PROGRAM Control_FBD
VAR

	timeStop: BOOL;
END_VAR

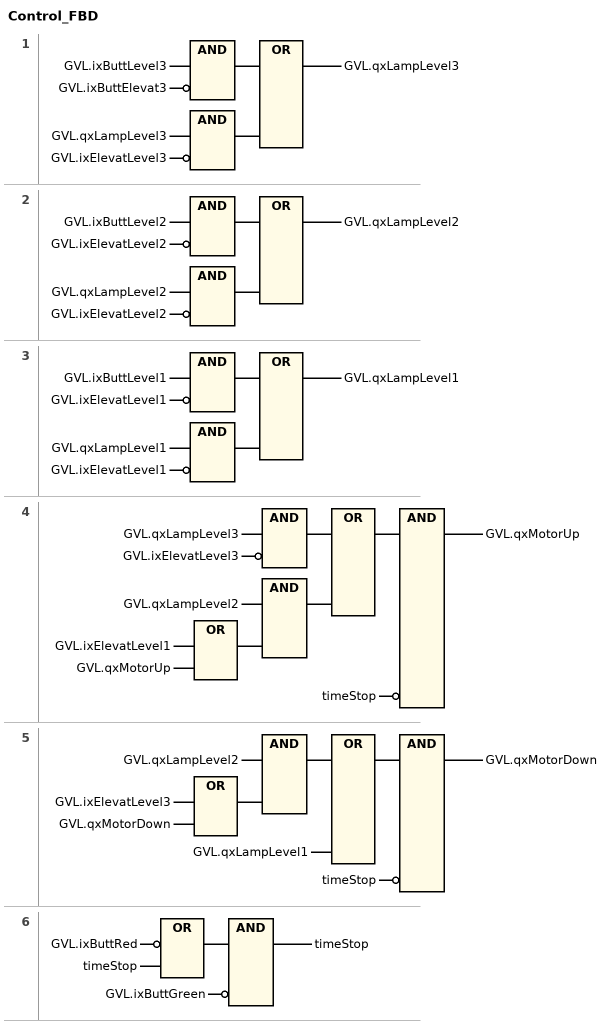
// NETWORK 1
GVL.qxLampLevel3 := GVL.ixButtLevel3 AND NOT GVL.ixButtElevat3 OR GVL.qxLampLevel3 AND NOT GVL.ixElevatLevel3;

// NETWORK 2
GVL.qxLampLevel2 := GVL.ixButtLevel2 AND NOT GVL.ixElevatLevel2 OR GVL.qxLampLevel2 AND NOT GVL.ixElevatLevel2;

// NETWORK 3
GVL.qxLampLevel1 := GVL.ixButtLevel1 AND NOT GVL.ixElevatLevel1 OR GVL.qxLampLevel1 AND NOT GVL.ixElevatLevel1;

// NETWORK 4
GVL.qxMotorUp := (GVL.qxLampLevel3 AND NOT GVL.ixElevatLevel3 OR GVL.qxLampLevel2 AND (GVL.ixElevatLevel1 OR GVL.qxMotorUp)) AND NOT timeStop;

// NETWORK 5
GVL.qxMotorDown := (GVL.qxLampLevel2 AND (GVL.ixElevatLevel3 OR GVL.qxMotorDown) OR GVL.qxLampLevel1) AND NOT timeStop;

// NETWORK 6
timeStop := (NOT GVL.ixButtRed OR timeStop) AND NOT GVL.ixButtGreen;

END_PROGRAM

(* stored: Version 1.1.0.1, ProductVersion 3.1.4024.12
   POU Control_FBD: Id {912119c4-f197-4ac1-96d5-56b57bc2b241}, SpecialFunc None *)
